// TIA Portal V17 export
// export: Created 2023-04-11T09:33:43.4785962Z, ExportSetting WithDefaults, DisplayName Totally Integrated Automation Portal, DisplayVersion V17 Update 3, DisplayName TIA Portal Openness, DisplayVersion V17 Update 3, DisplayName TIA Portal Version Control Interface, DisplayVersion V17, DisplayName SINAMICS Startdrive Advanced, DisplayVersion V17 Update2, DisplayName SINAMICS Startdrive G130, G150, S120, S150, SINAMICS MV, S210, DisplayVersion V17 Update2, DisplayName SINAMICS Startdrive G110M, G120, G120C, G120D, G120P, G115D, DisplayVersion V17 Update2, DisplayName STEP 7 Professional, DisplayVersion V17 Update 3, DisplayName STEP 7 Safety, DisplayVersion V17, DisplayName WinCC UA Professional, DisplayVersion V17 Update 3
FUNCTION "CON4DELIM_1" : Void   // FC45, LAD
{ S7_Optimized_Access := 'TRUE' }
VERSION : 0.1
// stored: AutoNumber true, IsIECCheckEnabled false, SetENOAutomatically false, UDAEnableTagReadback false
   VAR_IN_OUT
      Line : "t_LString";
      Delim : String;
      Part_1 : String;
      Part_2 : String;
      Part_3 : String;
      Part_4 : String;
   END_VAR
   VAR_TEMP   // added for the SCL form of the ladder/FBD networks
      _w1 : Bool;
      _w2 : Bool;
      _w3 : Bool;
      _w4 : Bool;
      _w5 : Bool;
      _w6 : Bool;
      _w7 : Bool;
   END_VAR
BEGIN

REGION Network 1: Line := Line + Part_1 + Delim + Part_2 + Delim + Part_3 + Delim + Part_4 + Delim
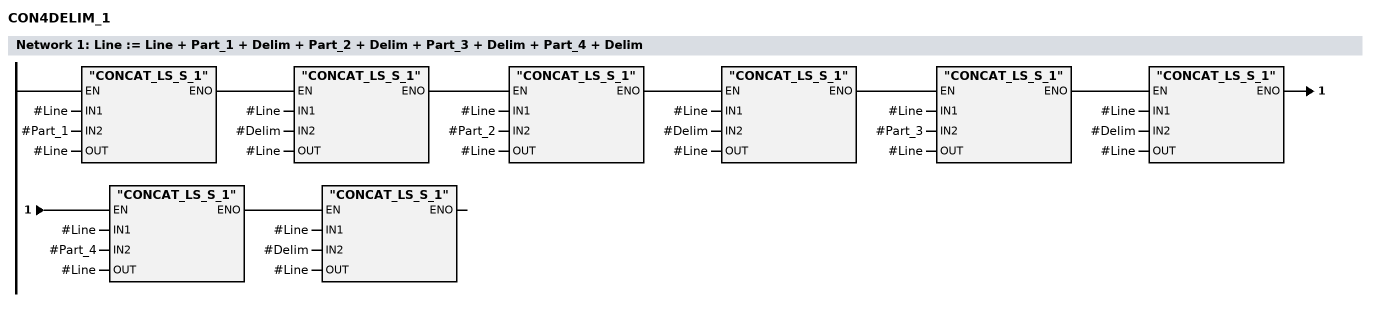
   RUNG wire#powerrail
      "CONCAT_LS_S_1"(IN1 := #Line, IN2 := #Part_1, OUT := #Line)
      "CONCAT_LS_S_1"(IN1 := #Line, IN2 := #Delim, OUT := #Line)
      "CONCAT_LS_S_1"(IN1 := #Line, IN2 := #Part_2, OUT := #Line)
      "CONCAT_LS_S_1"(IN1 := #Line, IN2 := #Delim, OUT := #Line)
      "CONCAT_LS_S_1"(IN1 := #Line, IN2 := #Part_3, OUT := #Line)
      "CONCAT_LS_S_1"(IN1 := #Line, IN2 := #Delim, OUT := #Line)
      "CONCAT_LS_S_1"(IN1 := #Line, IN2 := #Part_4, OUT := #Line)
      "CONCAT_LS_S_1"(IN1 := #Line, IN2 := #Delim, OUT := #Line)
   END_RUNG
   // the same network as SCL:
   "CONCAT_LS_S_1"(IN1 := #Line, IN2 := #Part_1, OUT := #Line, ENO => #_w1);
   "CONCAT_LS_S_1"(EN := #_w1, IN1 := #Line, IN2 := #Delim, OUT := #Line, ENO => #_w2);
   "CONCAT_LS_S_1"(EN := #_w2, IN1 := #Line, IN2 := #Part_2, OUT := #Line, ENO => #_w3);
   "CONCAT_LS_S_1"(EN := #_w3, IN1 := #Line, IN2 := #Delim, OUT := #Line, ENO => #_w4);
   "CONCAT_LS_S_1"(EN := #_w4, IN1 := #Line, IN2 := #Part_3, OUT := #Line, ENO => #_w5);
   "CONCAT_LS_S_1"(EN := #_w5, IN1 := #Line, IN2 := #Delim, OUT := #Line, ENO => #_w6);
   "CONCAT_LS_S_1"(EN := #_w6, IN1 := #Line, IN2 := #Part_4, OUT := #Line, ENO => #_w7);
   IF #_w7 THEN "CONCAT_LS_S_1"(IN1 := #Line, IN2 := #Delim, OUT := #Line); END_IF;
END_REGION
END_FUNCTION
